// Block: DEBUG_MES_Send_Msg_1XX

DATA_BLOCK DEBUG_MES_Send_Msg_1XX
VERSION : 0.1
   NON_RETAIN
   VAR
      MSG101 : Struct
         ABILITA_FC : Bool;
         EXE : Bool;
         RETVAL : DInt;
         Err : "MES_Err_&_Msg";
      END_STRUCT;
      MSG102 : Struct
         ABILITA_FC : Bool;
         EXE : Bool;
         RETVAL : DInt;
         Err : "MES_Err_&_Msg";
         MSG102 : Struct
            ABILITA_FC : Bool;
            EXE : Bool;
            RETVAL : DInt;
            Err : "MES_Err_&_Msg";
         END_STRUCT;
      END_STRUCT;
      TEST_FUN_BUFFER : Struct
         ABILITA_FC : Bool;
         RETVAL : DInt;
         lastId : DInt;
         Index : Int;
         Msg : MES_Msg;
         Evaluate_FULL : Bool;
         ClearGap : Bool;
         Push : Bool;
         Pop : Bool;
      END_STRUCT;
   END_VAR

BEGIN
   // No initialization required
END_DATA_BLOCK
